FUNCTION_BLOCK FB_InitDriveRefs
VAR_IN_OUT
	stCoE	:	ST_ElmoGDCBellCoEParams;
END_VAR
VAR_INPUT
END_VAR
VAR_OUTPUT
END_VAR
VAR
	
END_VAR

stCoE.stDriveRef.sNetId := F_CreateAmsNetId(gAmsNetIDEcatMaster1);
stCoE.stDriveRef.nDriveNo := stCoE.stPlcDriveRef.nDriveNo;
stCoE.stDriveRef.nDriveType := stCoE.stPlcDriveRef.nDriveType;
stCoE.stDriveRef.nSlaveAddr := stCoE.stPlcDriveRef.nSlaveAddr;

stCoE.AmsID := stCoE.stDriveRef.sNetId;
stCoE.nSlave := stCoE.stDriveRef.nSlaveAddr;

END_FUNCTION_BLOCK

(* stored: Version 1.1.0.1, ProductVersion 3.1.4024.6
   POU FB_InitDriveRefs: Id {f3c962b6-24fa-4ee7-ad86-91ec786ae7e0}, SpecialFunc None *)
